(* IEC 61131-3 sources: material-handling-micro-cell/plc, 14 files *)

(* ---- FB_AlarmManager.st ---- *)
// ==========================================
// ALARM MANAGER MODULE FOR MHMC-01
// File: FB_AlarmManager.st
// Standard: IEC 61131-3 Structured Text
// Purpose: Alarm categorisation, acknowledgement, and stack light control.
// ==========================================

TYPE E_AlarmManagerState :
(
    ALARM_MGR_UNINITIALISED := 0,
    ALARM_MGR_NORMAL        := 10,
    ALARM_MGR_WARNING       := 20,
    ALARM_MGR_FAULT         := 30,
    ALARM_MGR_ABORT         := 900
) INT;
END_TYPE

TYPE E_MHMCAlarmCode :
(
    ALARM_NONE        := 0,
    ALARM_GENERAL_JAM := 100,
    ALARM_DIVERTER_1  := 200,
    ALARM_DIVERTER_2  := 210,
    ALARM_AIR_PRESSURE:= 300,
    ALARM_VFD_FAULT   := 400,
    ALARM_ESTOP       := 1000
) INT;
END_TYPE

TYPE ST_AlarmManagerConfig :
STRUCT
    rFlashPeriod_s : REAL; // Stack light flash interval.
END_STRUCT
END_TYPE

TYPE ST_AlarmManagerInput :
STRUCT
    xSafetyLoopOK       : BOOL;          // Safety relay input.
    xAirPressureOK      : BOOL;          // Pneumatic pressure healthy.
    xVfdFault           : BOOL;          // Conveyor drive fault.
    xJamAlarm           : BOOL;          // Jam detector alarm.
    xJamWarning         : BOOL;          // Jam detector pre-alarm.
    xDiverter1Faulted   : BOOL;          // Diverter 1 fault.
    xDiverter2Faulted   : BOOL;          // Diverter 2 fault.
    ePackMLState        : E_PackML_State; // Station state for light logic.
    xAcknowledge        : BOOL;          // HMI/SCADA alarm acknowledge.
    xReset              : BOOL;          // Alarm reset when root cause clear.
    rCycleTime_s        : REAL;          // PLC task interval for tests.
END_STRUCT
END_TYPE

TYPE ST_AlarmManagerOutput :
STRUCT
    xAnyAlarmActive     : BOOL;          // Aggregate active alarm.
    xAnyUnacked         : BOOL;          // Active or latched unacknowledged alarm.
    eActiveAlarmCode    : E_MHMCAlarmCode; // Highest-priority active alarm.
    uiSeverity          : UINT;          // OPC UA AlarmCondition severity 1..1000.
    xGeneralJamAlarm    : BOOL;          // OPC UA GeneralJamAlarm active state.
    xDiverter1Alarm     : BOOL;          // OPC UA Diverter1Fault active state.
    xDiverter2Alarm     : BOOL;          // OPC UA Diverter2Fault active state.
    xEStopAlarm         : BOOL;          // OPC UA EStopTripped active state.
    xStackGreen         : BOOL;          // Run indicator.
    xStackYellow        : BOOL;          // Warning/held indicator.
    xStackRed           : BOOL;          // Abort/fault indicator.
    xSounder            : BOOL;          // Audible alarm output.
    sActiveMessage      : STRING(80);    // Alarm text for SCADA.
END_STRUCT
END_TYPE

TYPE ST_AlarmManagerContext :
STRUCT
    eState          : E_AlarmManagerState;
    xInitialized    : BOOL;
    xAckLatched     : BOOL;
    xFlashState     : BOOL;
    rFlashElapsed_s : REAL;
END_STRUCT
END_TYPE

FUNCTION F_AlarmManager_Init : BOOL
VAR_INPUT
    stConfig : ST_AlarmManagerConfig;
END_VAR
VAR_IN_OUT
    stContext : ST_AlarmManagerContext;
    stOut     : ST_AlarmManagerOutput;
END_VAR

// Initialisation function. Clears latched acknowledgement and drives indicators safe.
stContext.eState := E_AlarmManagerState.ALARM_MGR_NORMAL;
stContext.xInitialized := TRUE;
stContext.xAckLatched := FALSE;
stContext.xFlashState := FALSE;
stContext.rFlashElapsed_s := 0.0;

stOut.xAnyAlarmActive := FALSE;
stOut.xAnyUnacked := FALSE;
stOut.eActiveAlarmCode := E_MHMCAlarmCode.ALARM_NONE;
stOut.uiSeverity := 0;
stOut.xGeneralJamAlarm := FALSE;
stOut.xDiverter1Alarm := FALSE;
stOut.xDiverter2Alarm := FALSE;
stOut.xEStopAlarm := FALSE;
stOut.xStackGreen := FALSE;
stOut.xStackYellow := FALSE;
stOut.xStackRed := FALSE;
stOut.xSounder := FALSE;
stOut.sActiveMessage := 'Alarm manager initialised';

F_AlarmManager_Init := TRUE;
END_FUNCTION

FUNCTION F_AlarmManager_Cyclic : BOOL
VAR_INPUT
    stIn     : ST_AlarmManagerInput;
    stConfig : ST_AlarmManagerConfig;
END_VAR
VAR_IN_OUT
    stContext : ST_AlarmManagerContext;
    stOut     : ST_AlarmManagerOutput;
END_VAR

// Cyclic execution function. Highest severity wins; acknowledgement is separated from reset.
stContext.rFlashElapsed_s := stContext.rFlashElapsed_s + stIn.rCycleTime_s;
IF stContext.rFlashElapsed_s >= stConfig.rFlashPeriod_s THEN
    stContext.xFlashState := NOT stContext.xFlashState;
    stContext.rFlashElapsed_s := 0.0;
END_IF;

stOut.xGeneralJamAlarm := stIn.xJamAlarm;
stOut.xDiverter1Alarm := stIn.xDiverter1Faulted;
stOut.xDiverter2Alarm := stIn.xDiverter2Faulted;
stOut.xEStopAlarm := NOT stIn.xSafetyLoopOK;
stOut.xAnyAlarmActive := stOut.xGeneralJamAlarm
                         OR stOut.xDiverter1Alarm
                         OR stOut.xDiverter2Alarm
                         OR stOut.xEStopAlarm
                         OR stIn.xVfdFault
                         OR NOT stIn.xAirPressureOK;

IF stIn.xAcknowledge THEN
    stContext.xAckLatched := TRUE;
END_IF;
IF stIn.xReset AND NOT stOut.xAnyAlarmActive THEN
    stContext.xAckLatched := FALSE;
END_IF;

IF NOT stContext.xInitialized THEN
    stContext.eState := E_AlarmManagerState.ALARM_MGR_UNINITIALISED;
    stOut.eActiveAlarmCode := E_MHMCAlarmCode.ALARM_NONE;
    stOut.uiSeverity := 0;
    stOut.sActiveMessage := 'Alarm manager not initialised';
ELSIF NOT stIn.xSafetyLoopOK THEN
    stContext.eState := E_AlarmManagerState.ALARM_MGR_ABORT;
    stOut.eActiveAlarmCode := E_MHMCAlarmCode.ALARM_ESTOP;
    stOut.uiSeverity := 1000;
    stOut.sActiveMessage := 'Emergency stop circuit tripped';
ELSIF stIn.xDiverter1Faulted THEN
    stContext.eState := E_AlarmManagerState.ALARM_MGR_FAULT;
    stOut.eActiveAlarmCode := E_MHMCAlarmCode.ALARM_DIVERTER_1;
    stOut.uiSeverity := 900;
    stOut.sActiveMessage := 'Diverter 1 pneumatic actuator fault';
ELSIF stIn.xDiverter2Faulted THEN
    stContext.eState := E_AlarmManagerState.ALARM_MGR_FAULT;
    stOut.eActiveAlarmCode := E_MHMCAlarmCode.ALARM_DIVERTER_2;
    stOut.uiSeverity := 900;
    stOut.sActiveMessage := 'Diverter 2 pneumatic actuator fault';
ELSIF stIn.xJamAlarm THEN
    stContext.eState := E_AlarmManagerState.ALARM_MGR_FAULT;
    stOut.eActiveAlarmCode := E_MHMCAlarmCode.ALARM_GENERAL_JAM;
    stOut.uiSeverity := 800;
    stOut.sActiveMessage := 'Package jam detected on main conveyor';
ELSIF NOT stIn.xAirPressureOK THEN
    stContext.eState := E_AlarmManagerState.ALARM_MGR_FAULT;
    stOut.eActiveAlarmCode := E_MHMCAlarmCode.ALARM_AIR_PRESSURE;
    stOut.uiSeverity := 700;
    stOut.sActiveMessage := 'Pneumatic pressure below permissive threshold';
ELSIF stIn.xVfdFault THEN
    stContext.eState := E_AlarmManagerState.ALARM_MGR_FAULT;
    stOut.eActiveAlarmCode := E_MHMCAlarmCode.ALARM_VFD_FAULT;
    stOut.uiSeverity := 700;
    stOut.sActiveMessage := 'Conveyor VFD fault active';
ELSIF stIn.xJamWarning OR (stIn.ePackMLState = E_PackML_State.HELD) THEN
    stContext.eState := E_AlarmManagerState.ALARM_MGR_WARNING;
    stOut.eActiveAlarmCode := E_MHMCAlarmCode.ALARM_NONE;
    stOut.uiSeverity := 300;
    stOut.sActiveMessage := 'Cell warning or held state active';
ELSE
    stContext.eState := E_AlarmManagerState.ALARM_MGR_NORMAL;
    stOut.eActiveAlarmCode := E_MHMCAlarmCode.ALARM_NONE;
    stOut.uiSeverity := 0;
    stOut.sActiveMessage := 'No active alarms';
END_IF;

stOut.xAnyUnacked := stOut.xAnyAlarmActive AND NOT stContext.xAckLatched;
stOut.xStackGreen := (stIn.ePackMLState = E_PackML_State.EXECUTE) AND NOT stOut.xAnyAlarmActive;
stOut.xStackYellow := stContext.xFlashState
                      AND ((stContext.eState = E_AlarmManagerState.ALARM_MGR_WARNING)
                           OR stIn.xJamWarning
                           OR stIn.xJamAlarm);
stOut.xStackRed := stOut.xEStopAlarm
                   OR (stContext.eState = E_AlarmManagerState.ALARM_MGR_FAULT)
                   OR (stContext.eState = E_AlarmManagerState.ALARM_MGR_ABORT);
stOut.xSounder := stOut.xAnyUnacked AND (stOut.uiSeverity >= 800);

F_AlarmManager_Cyclic := stContext.xInitialized;
END_FUNCTION

FUNCTION_BLOCK FB_AlarmManager
VAR_INPUT
    stIn     : ST_AlarmManagerInput;  // Typed symbolic inputs.
    stConfig : ST_AlarmManagerConfig; // Testable alarm configuration.
    xInit    : BOOL;                  // Pulse to re-run initialisation.
END_VAR
VAR_OUTPUT
    stOut        : ST_AlarmManagerOutput; // Typed symbolic outputs.
    eState       : E_AlarmManagerState;   // Exposed module state.
    xInitialized : BOOL;                  // Module initialisation complete.
END_VAR
VAR
    stContext : ST_AlarmManagerContext;
    xInitLast : BOOL;
END_VAR

IF (NOT stContext.xInitialized) OR (xInit AND NOT xInitLast) THEN
    F_AlarmManager_Init(stConfig := stConfig, stContext := stContext, stOut := stOut);
END_IF;

F_AlarmManager_Cyclic(stIn := stIn, stConfig := stConfig, stContext := stContext, stOut := stOut);

eState := stContext.eState;
xInitialized := stContext.xInitialized;
xInitLast := xInit;
END_FUNCTION_BLOCK

(* ---- FB_DiverterController.st ---- *)
// ==========================================
// DIVERTER CONTROLLER MODULE FOR MHMC-01
// File: FB_DiverterController.st
// Standard: IEC 61131-3 Structured Text
// Purpose: Pneumatic pusher sequencing for Diverter 1 and Diverter 2.
// ==========================================

TYPE E_DiverterControllerState :
(
    DIVERTER_UNINITIALISED := 0,
    DIVERTER_HOME          := 10,
    DIVERTER_EXTENDING     := 20,
    DIVERTER_WORK          := 30,
    DIVERTER_VERIFY        := 40,
    DIVERTER_RETRACTING    := 50,
    DIVERTER_FAULT         := 900
) INT;
END_TYPE

TYPE ST_DiverterControllerConfig :
STRUCT
    tActuatorName          : STRING(40); // Symbolic device name for diagnostics.
    rExtendTimeout_s       : REAL;       // Max time to reach work switch.
    rRetractTimeout_s      : REAL;       // Max time to return home.
    rWorkDwell_s           : REAL;       // Hold time after work switch.
    rVerificationTimeout_s : REAL;       // Max time to see lane PE confirmation.
END_STRUCT
END_TYPE

TYPE ST_DiverterControllerInput :
STRUCT
    xAutoEnable          : BOOL; // True when PackML EXECUTE permits automatic firing.
    xExtendRequest       : BOOL; // Routing sequence asks this diverter to fire.
    xManualExtend        : BOOL; // Maintenance/manual symbolic override.
    xHomeSensor          : BOOL; // LSx_Home magnetic switch.
    xWorkSensor          : BOOL; // LSx_Work magnetic switch.
    xVerificationSensor  : BOOL; // PE4 or PE5 lane confirmation.
    xResetFault          : BOOL; // Reset local actuator fault.
    rCycleTime_s         : REAL; // PLC task interval for test harness.
END_STRUCT
END_TYPE

TYPE ST_DiverterControllerOutput :
STRUCT
    xCommandExtend       : BOOL; // Symbolic solenoid command. Bind externally to field I/O.
    xBusy                : BOOL; // Actuator sequence active.
    xDone                : BOOL; // One-cycle sequence complete.
    xFaulted             : BOOL; // Travel or verification timeout.
    xHome                : BOOL; // Mirrored home switch.
    xWork                : BOOL; // Mirrored work switch.
    xVerified            : BOOL; // Lane verification latched for this cycle.
    uiFaultCode          : UINT; // 0 none, 1 extend, 2 retract, 3 verify.
    sStatusText          : STRING(80);
END_STRUCT
END_TYPE

TYPE ST_DiverterControllerContext :
STRUCT
    eState               : E_DiverterControllerState;
    xInitialized         : BOOL;
    xRequestLast         : BOOL;
    xDoneLatch           : BOOL;
    rStateElapsed_s      : REAL;
END_STRUCT
END_TYPE

FUNCTION F_DiverterController_Init : BOOL
VAR_INPUT
    stConfig : ST_DiverterControllerConfig;
END_VAR
VAR_IN_OUT
    stContext : ST_DiverterControllerContext;
    stOut     : ST_DiverterControllerOutput;
END_VAR

// Initialisation function. De-energises the valve and clears local sequence memory.
stContext.eState := E_DiverterControllerState.DIVERTER_HOME;
stContext.xInitialized := TRUE;
stContext.xRequestLast := FALSE;
stContext.xDoneLatch := FALSE;
stContext.rStateElapsed_s := 0.0;

stOut.xCommandExtend := FALSE;
stOut.xBusy := FALSE;
stOut.xDone := FALSE;
stOut.xFaulted := FALSE;
stOut.xHome := FALSE;
stOut.xWork := FALSE;
stOut.xVerified := FALSE;
stOut.uiFaultCode := 0;
stOut.sStatusText := 'Diverter controller initialised';

F_DiverterController_Init := TRUE;
END_FUNCTION

FUNCTION F_DiverterController_Cyclic : BOOL
VAR_INPUT
    stIn     : ST_DiverterControllerInput;
    stConfig : ST_DiverterControllerConfig;
END_VAR
VAR_IN_OUT
    stContext : ST_DiverterControllerContext;
    stOut     : ST_DiverterControllerOutput;
END_VAR
VAR
    xFireRequest : BOOL;
END_VAR

// Cyclic execution function. Sequence states are deterministic and unit-test friendly.
IF stIn.rCycleTime_s > 0.0 THEN
    stContext.rStateElapsed_s := stContext.rStateElapsed_s + stIn.rCycleTime_s;
END_IF;

stOut.xDone := FALSE;
stOut.xHome := stIn.xHomeSensor;
stOut.xWork := stIn.xWorkSensor;
xFireRequest := ((stIn.xAutoEnable AND stIn.xExtendRequest) OR stIn.xManualExtend);

IF stIn.xResetFault THEN
    stOut.xFaulted := FALSE;
    stOut.uiFaultCode := 0;
    stOut.xVerified := FALSE;
    stContext.eState := E_DiverterControllerState.DIVERTER_HOME;
    stContext.rStateElapsed_s := 0.0;
END_IF;

IF NOT stContext.xInitialized THEN
    stContext.eState := E_DiverterControllerState.DIVERTER_UNINITIALISED;
    stOut.xFaulted := TRUE;
    stOut.uiFaultCode := 99;
ELSIF stOut.xFaulted THEN
    stContext.eState := E_DiverterControllerState.DIVERTER_FAULT;
ELSIF xFireRequest AND NOT stContext.xRequestLast
      AND (stContext.eState = E_DiverterControllerState.DIVERTER_HOME) THEN
    stContext.eState := E_DiverterControllerState.DIVERTER_EXTENDING;
    stContext.rStateElapsed_s := 0.0;
    stOut.xVerified := FALSE;
ELSIF stContext.eState = E_DiverterControllerState.DIVERTER_EXTENDING THEN
    IF stIn.xWorkSensor THEN
        stContext.eState := E_DiverterControllerState.DIVERTER_WORK;
        stContext.rStateElapsed_s := 0.0;
    ELSIF stContext.rStateElapsed_s >= stConfig.rExtendTimeout_s THEN
        stOut.xFaulted := TRUE;
        stOut.uiFaultCode := 1;
    END_IF;
ELSIF stContext.eState = E_DiverterControllerState.DIVERTER_WORK THEN
    IF stContext.rStateElapsed_s >= stConfig.rWorkDwell_s THEN
        stContext.eState := E_DiverterControllerState.DIVERTER_VERIFY;
        stContext.rStateElapsed_s := 0.0;
    END_IF;
ELSIF stContext.eState = E_DiverterControllerState.DIVERTER_VERIFY THEN
    IF stIn.xVerificationSensor THEN
        stOut.xVerified := TRUE;
        stContext.eState := E_DiverterControllerState.DIVERTER_RETRACTING;
        stContext.rStateElapsed_s := 0.0;
    ELSIF stContext.rStateElapsed_s >= stConfig.rVerificationTimeout_s THEN
        stOut.xFaulted := TRUE;
        stOut.uiFaultCode := 3;
    END_IF;
ELSIF stContext.eState = E_DiverterControllerState.DIVERTER_RETRACTING THEN
    IF stIn.xHomeSensor THEN
        stContext.eState := E_DiverterControllerState.DIVERTER_HOME;
        stContext.rStateElapsed_s := 0.0;
        stOut.xDone := TRUE;
    ELSIF stContext.rStateElapsed_s >= stConfig.rRetractTimeout_s THEN
        stOut.xFaulted := TRUE;
        stOut.uiFaultCode := 2;
    END_IF;
ELSE
    stContext.eState := E_DiverterControllerState.DIVERTER_HOME;
END_IF;

stOut.xCommandExtend := (stContext.eState = E_DiverterControllerState.DIVERTER_EXTENDING)
                        OR (stContext.eState = E_DiverterControllerState.DIVERTER_WORK)
                        OR (stContext.eState = E_DiverterControllerState.DIVERTER_VERIFY);
stOut.xBusy := (stContext.eState = E_DiverterControllerState.DIVERTER_EXTENDING)
               OR (stContext.eState = E_DiverterControllerState.DIVERTER_WORK)
               OR (stContext.eState = E_DiverterControllerState.DIVERTER_VERIFY)
               OR (stContext.eState = E_DiverterControllerState.DIVERTER_RETRACTING);

IF stOut.xFaulted THEN
    stOut.xCommandExtend := FALSE;
    stOut.xBusy := FALSE;
    stOut.sStatusText := 'Diverter fault active';
ELSIF stOut.xBusy THEN
    stOut.sStatusText := 'Diverter sequence active';
ELSE
    stOut.sStatusText := 'Diverter ready at home';
END_IF;

stContext.xRequestLast := xFireRequest;
F_DiverterController_Cyclic := stContext.xInitialized;
END_FUNCTION

FUNCTION_BLOCK FB_DiverterController
VAR_INPUT
    stIn     : ST_DiverterControllerInput;  // Typed symbolic inputs.
    stConfig : ST_DiverterControllerConfig; // Testable timing configuration.
    xInit    : BOOL;                        // Pulse to re-run initialisation.
END_VAR
VAR_OUTPUT
    stOut        : ST_DiverterControllerOutput; // Typed symbolic outputs.
    eState       : E_DiverterControllerState;   // Exposed module state.
    xInitialized : BOOL;                        // Module initialisation complete.
END_VAR
VAR
    stContext : ST_DiverterControllerContext;
    xInitLast : BOOL;
END_VAR

IF (NOT stContext.xInitialized) OR (xInit AND NOT xInitLast) THEN
    F_DiverterController_Init(stConfig := stConfig, stContext := stContext, stOut := stOut);
END_IF;

F_DiverterController_Cyclic(stIn := stIn, stConfig := stConfig, stContext := stContext, stOut := stOut);

eState := stContext.eState;
xInitialized := stContext.xInitialized;
xInitLast := xInit;
END_FUNCTION_BLOCK

(* ---- FB_HistorianConnector.st ---- *)
// ==========================================
// HISTORIAN CONNECTOR MODULE FOR MHMC-01
// File: FB_HistorianConnector.st
// Standard: IEC 61131-3 Structured Text
// Purpose: PLC-side historian publish health and sampling handshake skeleton.
// ==========================================

TYPE E_HistorianConnectorState :
(
    HIST_UNINITIALISED := 0,
    HIST_DISABLED      := 10,
    HIST_CONNECTING    := 20,
    HIST_CONNECTED     := 30,
    HIST_PUBLISHING    := 40,
    HIST_BACKOFF       := 50,
    HIST_FAULTED       := 900
) INT;
END_TYPE

TYPE ST_HistorianConnectorConfig :
STRUCT
    tOpcUaNamespaceUri      : STRING(120); // Namespace URI, not an address binding.
    rSamplePeriod_s         : REAL;        // Historian sample strobe period.
    rHeartbeatTimeout_s     : REAL;        // Max time without collector heartbeat.
    uiMaxMissedHeartbeats   : UINT;        // Fault threshold.
END_STRUCT
END_TYPE

TYPE ST_HistorianConnectorInput :
STRUCT
    xEnable              : BOOL;               // Enable historian handshake.
    xOpcUaServerReady    : BOOL;               // OPC UA server namespace ready.
    xCollectorHeartbeat  : BOOL;               // Telegraf/collector heartbeat bit.
    xLastWriteOK         : BOOL;               // Influx write success from collector.
    stConveyor           : ST_Conveyor_Status; // Conveyor telemetry source.
    stDiverter1          : ST_Diverter_Status; // Diverter 1 telemetry source.
    stDiverter2          : ST_Diverter_Status; // Diverter 2 telemetry source.
    udiTotalCount        : UDINT;              // KPI source.
    udiLaneACount        : UDINT;              // KPI source.
    udiLaneBCount        : UDINT;              // KPI source.
    udiRejectCount       : UDINT;              // KPI source.
    uiTotalJams          : UINT;               // KPI source.
    rOEE_percent         : REAL;               // KPI source.
    xActiveAlarm         : BOOL;               // Alarm/event source.
    sActiveAlarmMessage  : STRING(80);         // Alarm/event source.
    rCycleTime_s         : REAL;               // PLC task interval for tests.
END_STRUCT
END_TYPE

TYPE ST_HistorianConnectorOutput :
STRUCT
    xSubscribeEnable      : BOOL;       // Allows collector to subscribe/poll OPC UA.
    xSampleStrobe         : BOOL;       // One-cycle sample request.
    xHistorianHealthy     : BOOL;       // True when OPC UA and collector are healthy.
    xPublishConveyor      : BOOL;       // Sample conveyor_telemetry.
    xPublishDiverter      : BOOL;       // Sample diverter_telemetry.
    xPublishKPI           : BOOL;       // Sample cell_kpis.
    xPublishAlarm         : BOOL;       // Sample alarms_events.
    uiMissedHeartbeats    : UINT;       // Collector heartbeat misses.
    sNamespaceUri         : STRING(120); // OPC UA namespace exposed to collector.
    sMeasurementClass     : STRING(40);  // Current logical measurement group.
    sLineProtocolPayload  : STRING(255); // Skeleton payload contract for collector tests.
    sStatusText           : STRING(80);
END_STRUCT
END_TYPE

TYPE ST_HistorianConnectorContext :
STRUCT
    eState             : E_HistorianConnectorState;
    xInitialized       : BOOL;
    xHeartbeatLast     : BOOL;
    rSampleElapsed_s   : REAL;
    rHeartbeatElapsed_s: REAL;
END_STRUCT
END_TYPE

FUNCTION F_HistorianConnector_Init : BOOL
VAR_INPUT
    stConfig : ST_HistorianConnectorConfig;
END_VAR
VAR_IN_OUT
    stContext : ST_HistorianConnectorContext;
    stOut     : ST_HistorianConnectorOutput;
END_VAR

// Initialisation function. The actual OPC UA/Influx endpoints remain external configuration.
stContext.eState := E_HistorianConnectorState.HIST_DISABLED;
stContext.xInitialized := TRUE;
stContext.xHeartbeatLast := FALSE;
stContext.rSampleElapsed_s := 0.0;
stContext.rHeartbeatElapsed_s := 0.0;

stOut.xSubscribeEnable := FALSE;
stOut.xSampleStrobe := FALSE;
stOut.xHistorianHealthy := FALSE;
stOut.xPublishConveyor := FALSE;
stOut.xPublishDiverter := FALSE;
stOut.xPublishKPI := FALSE;
stOut.xPublishAlarm := FALSE;
stOut.uiMissedHeartbeats := 0;
stOut.sNamespaceUri := stConfig.tOpcUaNamespaceUri;
stOut.sMeasurementClass := 'none';
stOut.sLineProtocolPayload := '';
stOut.sStatusText := 'Historian connector initialised';

F_HistorianConnector_Init := TRUE;
END_FUNCTION

FUNCTION F_HistorianConnector_Cyclic : BOOL
VAR_INPUT
    stIn     : ST_HistorianConnectorInput;
    stConfig : ST_HistorianConnectorConfig;
END_VAR
VAR_IN_OUT
    stContext : ST_HistorianConnectorContext;
    stOut     : ST_HistorianConnectorOutput;
END_VAR
VAR
    xHeartbeatEdge : BOOL;
END_VAR

// Cyclic execution function. Provides deterministic sample strobes for Telegraf/SCADA.
stOut.xSampleStrobe := FALSE;
stOut.xPublishConveyor := FALSE;
stOut.xPublishDiverter := FALSE;
stOut.xPublishKPI := FALSE;
stOut.xPublishAlarm := FALSE;
stOut.sNamespaceUri := stConfig.tOpcUaNamespaceUri;

xHeartbeatEdge := stIn.xCollectorHeartbeat <> stContext.xHeartbeatLast;
IF xHeartbeatEdge THEN
    stContext.rHeartbeatElapsed_s := 0.0;
    stOut.uiMissedHeartbeats := 0;
ELSE
    stContext.rHeartbeatElapsed_s := stContext.rHeartbeatElapsed_s + stIn.rCycleTime_s;
END_IF;

IF stContext.rHeartbeatElapsed_s >= stConfig.rHeartbeatTimeout_s THEN
    stOut.uiMissedHeartbeats := stOut.uiMissedHeartbeats + 1;
    stContext.rHeartbeatElapsed_s := 0.0;
END_IF;

IF NOT stContext.xInitialized THEN
    stContext.eState := E_HistorianConnectorState.HIST_UNINITIALISED;
ELSIF NOT stIn.xEnable THEN
    stContext.eState := E_HistorianConnectorState.HIST_DISABLED;
ELSIF NOT stIn.xOpcUaServerReady THEN
    stContext.eState := E_HistorianConnectorState.HIST_CONNECTING;
ELSIF stOut.uiMissedHeartbeats >= stConfig.uiMaxMissedHeartbeats THEN
    stContext.eState := E_HistorianConnectorState.HIST_BACKOFF;
ELSIF NOT stIn.xLastWriteOK THEN
    stContext.eState := E_HistorianConnectorState.HIST_FAULTED;
ELSE
    stContext.eState := E_HistorianConnectorState.HIST_CONNECTED;
END_IF;

stOut.xSubscribeEnable := stIn.xEnable AND stIn.xOpcUaServerReady;
stOut.xHistorianHealthy := stOut.xSubscribeEnable
                           AND (stOut.uiMissedHeartbeats < stConfig.uiMaxMissedHeartbeats)
                           AND stIn.xLastWriteOK;

IF stOut.xHistorianHealthy THEN
    stContext.rSampleElapsed_s := stContext.rSampleElapsed_s + stIn.rCycleTime_s;
    IF stContext.rSampleElapsed_s >= stConfig.rSamplePeriod_s THEN
        stContext.rSampleElapsed_s := 0.0;
        stContext.eState := E_HistorianConnectorState.HIST_PUBLISHING;
        stOut.xSampleStrobe := TRUE;
        stOut.xPublishConveyor := TRUE;
        stOut.xPublishDiverter := TRUE;
        stOut.xPublishKPI := TRUE;
        stOut.xPublishAlarm := stIn.xActiveAlarm;
    END_IF;
END_IF;

IF stOut.xPublishAlarm THEN
    stOut.sMeasurementClass := 'alarms_events';
    stOut.sLineProtocolPayload := 'alarms_events active=true';
ELSIF stOut.xPublishKPI THEN
    stOut.sMeasurementClass := 'cell_kpis';
    stOut.sLineProtocolPayload := 'cell_kpis sample=true';
ELSIF stOut.xPublishDiverter THEN
    stOut.sMeasurementClass := 'diverter_telemetry';
    stOut.sLineProtocolPayload := 'diverter_telemetry sample=true';
ELSIF stOut.xPublishConveyor THEN
    stOut.sMeasurementClass := 'conveyor_telemetry';
    stOut.sLineProtocolPayload := 'conveyor_telemetry sample=true';
ELSE
    stOut.sMeasurementClass := 'idle';
    stOut.sLineProtocolPayload := '';
END_IF;

IF stOut.xHistorianHealthy THEN
    stOut.sStatusText := 'Historian connector healthy';
ELSE
    stOut.sStatusText := 'Historian connector waiting for healthy collector';
END_IF;

stContext.xHeartbeatLast := stIn.xCollectorHeartbeat;
F_HistorianConnector_Cyclic := stContext.xInitialized;
END_FUNCTION

FUNCTION_BLOCK FB_HistorianConnector
VAR_INPUT
    stIn     : ST_HistorianConnectorInput;  // Typed symbolic inputs.
    stConfig : ST_HistorianConnectorConfig; // Testable historian configuration.
    xInit    : BOOL;                        // Pulse to re-run initialisation.
END_VAR
VAR_OUTPUT
    stOut        : ST_HistorianConnectorOutput; // Typed symbolic outputs.
    eState       : E_HistorianConnectorState;   // Exposed module state.
    xInitialized : BOOL;                        // Module initialisation complete.
END_VAR
VAR
    stContext : ST_HistorianConnectorContext;
    xInitLast : BOOL;
END_VAR

IF (NOT stContext.xInitialized) OR (xInit AND NOT xInitLast) THEN
    F_HistorianConnector_Init(stConfig := stConfig, stContext := stContext, stOut := stOut);
END_IF;

F_HistorianConnector_Cyclic(stIn := stIn, stConfig := stConfig, stContext := stContext, stOut := stOut);

eState := stContext.eState;
xInitialized := stContext.xInitialized;
xInitLast := xInit;
END_FUNCTION_BLOCK

(* ---- FB_JamDetector.st ---- *)
// ==========================================
// JAM DETECTOR MODULE FOR MHMC-01
// File: FB_JamDetector.st
// Standard: IEC 61131-3 Structured Text
// Purpose: Dynamic PE1/PE2/PE3 blockage watchdogs.
// ==========================================

TYPE E_JamDetectorState :
(
    JAM_DET_UNINITIALISED := 0,
    JAM_DET_CLEAR         := 10,
    JAM_DET_MONITORING    := 20,
    JAM_DET_WARNING       := 30,
    JAM_DET_JAMMED        := 900
) INT;
END_TYPE

TYPE ST_JamDetectorConfig :
STRUCT
    rReferenceSpeed_mps : REAL; // Speed used for nominal 3.0 s FDS limit.
    rBaseJamLimit_s     : REAL; // Nominal jam threshold at reference speed.
    rMaximumJamLimit_s  : REAL; // Slow-speed upper watchdog bound.
    rWarningRatio       : REAL; // Warning before full jam, e.g. 0.80.
END_STRUCT
END_TYPE

TYPE ST_JamDetectorInput :
STRUCT
    xRawPE1            : BOOL; // PE1 infeed blocked.
    xRawPE2            : BOOL; // PE2 scan trigger blocked.
    xRawPE3            : BOOL; // PE3 diverter in-range blocked.
    xConveyorRunning   : BOOL; // Conveyor feedback.
    rConveyorSpeed_mps : REAL; // Conveyor feedback speed.
    xResetJam          : BOOL; // ResetJam RPC/HMI command.
    rCycleTime_s       : REAL; // PLC task interval for unit tests.
END_STRUCT
END_TYPE

TYPE ST_JamDetectorOutput :
STRUCT
    xJamAlarm          : BOOL; // Fault flag to StationController.
    xWarning           : BOOL; // Pre-alarm for HMI and beacon logic.
    xBeaconYellowFlash : BOOL; // Symbolic stack light request.
    uiJamSource        : UINT; // 0 none, 1 PE1, 2 PE2, 3 PE3.
    uiTotalJams        : UINT; // OPC UA KPI TotalJams node.
    rActiveLimit_s     : REAL; // Dynamic watchdog threshold in use.
    sStatusText        : STRING(80);
END_STRUCT
END_TYPE

TYPE ST_JamDetectorContext :
STRUCT
    eState          : E_JamDetectorState;
    xInitialized    : BOOL;
    xJamLatchedLast : BOOL;
    rPE1Blocked_s   : REAL;
    rPE2Blocked_s   : REAL;
    rPE3Blocked_s   : REAL;
END_STRUCT
END_TYPE

FUNCTION F_JamDetector_DynamicLimit_s : REAL
VAR_INPUT
    rConveyorSpeed_mps : REAL;
    stConfig           : ST_JamDetectorConfig;
END_VAR
VAR
    rLimit_s : REAL;
END_VAR

// Dynamic limit increases as conveyor speed drops. It is clamped for slow jog cases.
IF rConveyorSpeed_mps <= 0.01 THEN
    rLimit_s := stConfig.rMaximumJamLimit_s;
ELSE
    rLimit_s := stConfig.rBaseJamLimit_s * stConfig.rReferenceSpeed_mps / rConveyorSpeed_mps;
END_IF;

IF rLimit_s < stConfig.rBaseJamLimit_s THEN
    rLimit_s := stConfig.rBaseJamLimit_s;
END_IF;
IF rLimit_s > stConfig.rMaximumJamLimit_s THEN
    rLimit_s := stConfig.rMaximumJamLimit_s;
END_IF;

F_JamDetector_DynamicLimit_s := rLimit_s;
END_FUNCTION

FUNCTION F_JamDetector_Init : BOOL
VAR_INPUT
    stConfig : ST_JamDetectorConfig;
END_VAR
VAR_IN_OUT
    stContext : ST_JamDetectorContext;
    stOut     : ST_JamDetectorOutput;
END_VAR

// Initialisation function. Clears watchdog accumulators and alarm outputs.
stContext.eState := E_JamDetectorState.JAM_DET_CLEAR;
stContext.xInitialized := TRUE;
stContext.xJamLatchedLast := FALSE;
stContext.rPE1Blocked_s := 0.0;
stContext.rPE2Blocked_s := 0.0;
stContext.rPE3Blocked_s := 0.0;

stOut.xJamAlarm := FALSE;
stOut.xWarning := FALSE;
stOut.xBeaconYellowFlash := FALSE;
stOut.uiJamSource := 0;
stOut.uiTotalJams := 0;
stOut.rActiveLimit_s := stConfig.rBaseJamLimit_s;
stOut.sStatusText := 'Jam detector initialised';

F_JamDetector_Init := TRUE;
END_FUNCTION

FUNCTION F_JamDetector_Cyclic : BOOL
VAR_INPUT
    stIn     : ST_JamDetectorInput;
    stConfig : ST_JamDetectorConfig;
END_VAR
VAR_IN_OUT
    stContext : ST_JamDetectorContext;
    stOut     : ST_JamDetectorOutput;
END_VAR
VAR
    rWarnLimit_s : REAL;
    xAnyBlocked  : BOOL;
END_VAR

// Cyclic execution function. PE watchdogs are independent and symbolic.
stOut.rActiveLimit_s := F_JamDetector_DynamicLimit_s(rConveyorSpeed_mps := stIn.rConveyorSpeed_mps, stConfig := stConfig);
rWarnLimit_s := stOut.rActiveLimit_s * stConfig.rWarningRatio;
xAnyBlocked := stIn.xRawPE1 OR stIn.xRawPE2 OR stIn.xRawPE3;

IF stIn.xResetJam THEN
    stOut.xJamAlarm := FALSE;
    stOut.xWarning := FALSE;
    stOut.xBeaconYellowFlash := FALSE;
    stOut.uiJamSource := 0;
    stContext.rPE1Blocked_s := 0.0;
    stContext.rPE2Blocked_s := 0.0;
    stContext.rPE3Blocked_s := 0.0;
    stContext.eState := E_JamDetectorState.JAM_DET_CLEAR;
END_IF;

IF stIn.xConveyorRunning THEN
    IF stIn.xRawPE1 THEN
        stContext.rPE1Blocked_s := stContext.rPE1Blocked_s + stIn.rCycleTime_s;
    ELSE
        stContext.rPE1Blocked_s := 0.0;
    END_IF;

    IF stIn.xRawPE2 THEN
        stContext.rPE2Blocked_s := stContext.rPE2Blocked_s + stIn.rCycleTime_s;
    ELSE
        stContext.rPE2Blocked_s := 0.0;
    END_IF;

    IF stIn.xRawPE3 THEN
        stContext.rPE3Blocked_s := stContext.rPE3Blocked_s + stIn.rCycleTime_s;
    ELSE
        stContext.rPE3Blocked_s := 0.0;
    END_IF;
END_IF;

IF NOT stContext.xInitialized THEN
    stContext.eState := E_JamDetectorState.JAM_DET_UNINITIALISED;
ELSIF (stContext.rPE1Blocked_s >= stOut.rActiveLimit_s)
      OR (stContext.rPE2Blocked_s >= stOut.rActiveLimit_s)
      OR (stContext.rPE3Blocked_s >= stOut.rActiveLimit_s) THEN
    stContext.eState := E_JamDetectorState.JAM_DET_JAMMED;
    stOut.xJamAlarm := TRUE;
    IF stContext.rPE1Blocked_s >= stOut.rActiveLimit_s THEN
        stOut.uiJamSource := 1;
    ELSIF stContext.rPE2Blocked_s >= stOut.rActiveLimit_s THEN
        stOut.uiJamSource := 2;
    ELSE
        stOut.uiJamSource := 3;
    END_IF;
ELSIF (stContext.rPE1Blocked_s >= rWarnLimit_s)
      OR (stContext.rPE2Blocked_s >= rWarnLimit_s)
      OR (stContext.rPE3Blocked_s >= rWarnLimit_s) THEN
    stContext.eState := E_JamDetectorState.JAM_DET_WARNING;
    stOut.xWarning := TRUE;
ELSE
    stOut.xWarning := FALSE;
    IF xAnyBlocked AND stIn.xConveyorRunning THEN
        stContext.eState := E_JamDetectorState.JAM_DET_MONITORING;
    ELSE
        stContext.eState := E_JamDetectorState.JAM_DET_CLEAR;
    END_IF;
END_IF;

IF stOut.xJamAlarm AND NOT stContext.xJamLatchedLast THEN
    stOut.uiTotalJams := stOut.uiTotalJams + 1;
END_IF;

stOut.xBeaconYellowFlash := stOut.xWarning OR stOut.xJamAlarm;
IF stOut.xJamAlarm THEN
    stOut.sStatusText := 'Package jam detected on main conveyor';
ELSIF stOut.xWarning THEN
    stOut.sStatusText := 'Photoeye blocked near jam threshold';
ELSE
    stOut.sStatusText := 'Jam detector clear';
END_IF;

stContext.xJamLatchedLast := stOut.xJamAlarm;
F_JamDetector_Cyclic := stContext.xInitialized;
END_FUNCTION

FUNCTION_BLOCK FB_JamDetector
VAR_INPUT
    stIn     : ST_JamDetectorInput;  // Typed symbolic inputs.
    stConfig : ST_JamDetectorConfig; // Testable watchdog configuration.
    xInit    : BOOL;                 // Pulse to re-run initialisation.
END_VAR
VAR_OUTPUT
    stOut        : ST_JamDetectorOutput; // Typed symbolic outputs.
    eState       : E_JamDetectorState;   // Exposed module state.
    xInitialized : BOOL;                 // Module initialisation complete.
END_VAR
VAR
    stContext : ST_JamDetectorContext;
    xInitLast : BOOL;
END_VAR

IF (NOT stContext.xInitialized) OR (xInit AND NOT xInitLast) THEN
    F_JamDetector_Init(stConfig := stConfig, stContext := stContext, stOut := stOut);
END_IF;

F_JamDetector_Cyclic(stIn := stIn, stConfig := stConfig, stContext := stContext, stOut := stOut);

eState := stContext.eState;
xInitialized := stContext.xInitialized;
xInitLast := xInit;
END_FUNCTION_BLOCK

(* ---- FB_KPIService.st ---- *)
// ==========================================
// KPI SERVICE MODULE FOR MHMC-01
// File: FB_KPIService.st
// Standard: IEC 61131-3 Structured Text
// Purpose: Throughput counters and OEE calculation skeleton.
// ==========================================

TYPE E_KPIServiceState :
(
    KPI_UNINITIALISED := 0,
    KPI_IDLE          := 10,
    KPI_ACCUMULATING  := 20,
    KPI_HELD          := 30,
    KPI_RESETTING     := 40
) INT;
END_TYPE

TYPE ST_KPIServiceConfig :
STRUCT
    rPerformanceFactor : REAL; // FDS target sorting velocity efficiency, e.g. 0.96.
    rTargetRate_ppm    : REAL; // Target packages per minute for throughput trending.
END_STRUCT
END_TYPE

TYPE ST_KPIServiceInput :
STRUCT
    xPE4LaneA        : BOOL;          // Lane A verification sensor.
    xPE5LaneB        : BOOL;          // Lane B verification sensor.
    xPE6Reject       : BOOL;          // Reject verification sensor.
    ePackMLState     : E_PackML_State; // Station state for availability.
    xFaultDowntime   : BOOL;          // Fault/held downtime active.
    xResetCounters   : BOOL;          // KPI reset command.
    rCycleTime_s     : REAL;          // PLC task interval for tests.
END_STRUCT
END_TYPE

TYPE ST_KPIServiceOutput :
STRUCT
    udiTotalPackages     : UDINT; // Total package count.
    udiLaneAPackages     : UDINT; // Lane A count.
    udiLaneBPackages     : UDINT; // Lane B count.
    udiRejectPackages    : UDINT; // Reject count.
    rAvailability        : REAL;  // Execute / scheduled time.
    rPerformance         : REAL;  // Target sorting velocity efficiency.
    rQuality             : REAL;  // (Total - Reject) / Total.
    rOEE_percent         : REAL;  // Availability * Performance * Quality * 100.
    rThroughput_ppm      : REAL;  // Recent average from total/scheduled time.
    sStatusText          : STRING(80);
END_STRUCT
END_TYPE

TYPE ST_KPIServiceContext :
STRUCT
    eState            : E_KPIServiceState;
    xInitialized      : BOOL;
    xPE4Last          : BOOL;
    xPE5Last          : BOOL;
    xPE6Last          : BOOL;
    rExecuteTime_s    : REAL;
    rFaultDowntime_s  : REAL;
    rScheduledTime_s  : REAL;
END_STRUCT
END_TYPE

FUNCTION F_KPIService_Init : BOOL
VAR_INPUT
    stConfig : ST_KPIServiceConfig;
END_VAR
VAR_IN_OUT
    stContext : ST_KPIServiceContext;
    stOut     : ST_KPIServiceOutput;
END_VAR

// Initialisation function. Clears counters and restores default OEE factors.
stContext.eState := E_KPIServiceState.KPI_IDLE;
stContext.xInitialized := TRUE;
stContext.xPE4Last := FALSE;
stContext.xPE5Last := FALSE;
stContext.xPE6Last := FALSE;
stContext.rExecuteTime_s := 0.0;
stContext.rFaultDowntime_s := 0.0;
stContext.rScheduledTime_s := 0.0;

stOut.udiTotalPackages := 0;
stOut.udiLaneAPackages := 0;
stOut.udiLaneBPackages := 0;
stOut.udiRejectPackages := 0;
stOut.rAvailability := 1.0;
stOut.rPerformance := stConfig.rPerformanceFactor;
stOut.rQuality := 1.0;
stOut.rOEE_percent := stOut.rAvailability * stOut.rPerformance * stOut.rQuality * 100.0;
stOut.rThroughput_ppm := 0.0;
stOut.sStatusText := 'KPI service initialised';

F_KPIService_Init := TRUE;
END_FUNCTION

FUNCTION F_KPIService_Cyclic : BOOL
VAR_INPUT
    stIn     : ST_KPIServiceInput;
    stConfig : ST_KPIServiceConfig;
END_VAR
VAR_IN_OUT
    stContext : ST_KPIServiceContext;
    stOut     : ST_KPIServiceOutput;
END_VAR
VAR
    xPE4Rise : BOOL;
    xPE5Rise : BOOL;
    xPE6Rise : BOOL;
END_VAR

// Cyclic execution function. Sensor edges drive counters; PackML state drives availability.
IF stIn.xResetCounters THEN
    stContext.eState := E_KPIServiceState.KPI_RESETTING;
    stContext.rExecuteTime_s := 0.0;
    stContext.rFaultDowntime_s := 0.0;
    stContext.rScheduledTime_s := 0.0;
    stOut.udiTotalPackages := 0;
    stOut.udiLaneAPackages := 0;
    stOut.udiLaneBPackages := 0;
    stOut.udiRejectPackages := 0;
END_IF;

xPE4Rise := stIn.xPE4LaneA AND NOT stContext.xPE4Last;
xPE5Rise := stIn.xPE5LaneB AND NOT stContext.xPE5Last;
xPE6Rise := stIn.xPE6Reject AND NOT stContext.xPE6Last;

IF xPE4Rise THEN
    stOut.udiLaneAPackages := stOut.udiLaneAPackages + 1;
    stOut.udiTotalPackages := stOut.udiTotalPackages + 1;
END_IF;
IF xPE5Rise THEN
    stOut.udiLaneBPackages := stOut.udiLaneBPackages + 1;
    stOut.udiTotalPackages := stOut.udiTotalPackages + 1;
END_IF;
IF xPE6Rise THEN
    stOut.udiRejectPackages := stOut.udiRejectPackages + 1;
    stOut.udiTotalPackages := stOut.udiTotalPackages + 1;
END_IF;

IF stIn.ePackMLState = E_PackML_State.EXECUTE THEN
    stContext.eState := E_KPIServiceState.KPI_ACCUMULATING;
    stContext.rExecuteTime_s := stContext.rExecuteTime_s + stIn.rCycleTime_s;
    stContext.rScheduledTime_s := stContext.rScheduledTime_s + stIn.rCycleTime_s;
ELSIF stIn.xFaultDowntime OR (stIn.ePackMLState = E_PackML_State.HELD) THEN
    stContext.eState := E_KPIServiceState.KPI_HELD;
    stContext.rFaultDowntime_s := stContext.rFaultDowntime_s + stIn.rCycleTime_s;
    stContext.rScheduledTime_s := stContext.rScheduledTime_s + stIn.rCycleTime_s;
ELSE
    stContext.eState := E_KPIServiceState.KPI_IDLE;
END_IF;

IF stContext.rScheduledTime_s > 0.0 THEN
    stOut.rAvailability := stContext.rExecuteTime_s / stContext.rScheduledTime_s;
    stOut.rThroughput_ppm := UDINT_TO_REAL(stOut.udiTotalPackages) / (stContext.rScheduledTime_s / 60.0);
ELSE
    stOut.rAvailability := 1.0;
    stOut.rThroughput_ppm := 0.0;
END_IF;

stOut.rPerformance := stConfig.rPerformanceFactor;
IF stOut.udiTotalPackages > 0 THEN
    stOut.rQuality := (UDINT_TO_REAL(stOut.udiTotalPackages) - UDINT_TO_REAL(stOut.udiRejectPackages))
                      / UDINT_TO_REAL(stOut.udiTotalPackages);
ELSE
    stOut.rQuality := 1.0;
END_IF;

stOut.rOEE_percent := stOut.rAvailability * stOut.rPerformance * stOut.rQuality * 100.0;
stOut.sStatusText := 'KPI service calculated counters and OEE';

stContext.xPE4Last := stIn.xPE4LaneA;
stContext.xPE5Last := stIn.xPE5LaneB;
stContext.xPE6Last := stIn.xPE6Reject;
F_KPIService_Cyclic := stContext.xInitialized;
END_FUNCTION

FUNCTION_BLOCK FB_KPIService
VAR_INPUT
    stIn     : ST_KPIServiceInput;  // Typed symbolic inputs.
    stConfig : ST_KPIServiceConfig; // Testable KPI configuration.
    xInit    : BOOL;                // Pulse to re-run initialisation.
END_VAR
VAR_OUTPUT
    stOut        : ST_KPIServiceOutput; // Typed symbolic outputs.
    eState       : E_KPIServiceState;   // Exposed module state.
    xInitialized : BOOL;                // Module initialisation complete.
END_VAR
VAR
    stContext : ST_KPIServiceContext;
    xInitLast : BOOL;
END_VAR

IF (NOT stContext.xInitialized) OR (xInit AND NOT xInitLast) THEN
    F_KPIService_Init(stConfig := stConfig, stContext := stContext, stOut := stOut);
END_IF;

F_KPIService_Cyclic(stIn := stIn, stConfig := stConfig, stContext := stContext, stOut := stOut);

eState := stContext.eState;
xInitialized := stContext.xInitialized;
xInitLast := xInit;
END_FUNCTION_BLOCK

(* ---- FB_LineSupervisor.st ---- *)
// ==========================================
// LINE SUPERVISOR MODULE FOR MHMC-01
// File: FB_LineSupervisor.st
// Standard: IEC 61131-3 Structured Text
// Purpose: Cell-level command, mode, and recipe dispatch skeleton.
// ==========================================

TYPE E_LineSupervisorState :
(
    LINE_SUP_UNINITIALISED := 0,
    LINE_SUP_READY         := 10,
    LINE_SUP_RECIPE_LOAD   := 20,
    LINE_SUP_COMMANDING    := 30,
    LINE_SUP_FAULTED       := 900
) INT;
END_TYPE

TYPE ST_LineSupervisorConfig :
STRUCT
    rDefaultTargetSpeed_mps : REAL;       // Recipe default conveyor speed.
    rMinimumTargetSpeed_mps : REAL;       // Lower recipe validation bound.
    rMaximumTargetSpeed_mps : REAL;       // Upper recipe validation bound.
    sLaneAPattern           : STRING(40); // Symbolic barcode rule for Lane A.
    sLaneBPattern           : STRING(40); // Symbolic barcode rule for Lane B.
    sRejectPattern          : STRING(40); // Symbolic barcode rule for reject/default.
END_STRUCT
END_TYPE

TYPE ST_LineSupervisorInput :
STRUCT
    xStartCommand      : BOOL;          // HMI/OPC UA StartCell request.
    xStopCommand       : BOOL;          // HMI/OPC UA StopCell request.
    xResetCommand      : BOOL;          // HMI/OPC UA reset request.
    xHoldCommand       : BOOL;          // HMI/SCADA hold request.
    xUnholdCommand     : BOOL;          // HMI/SCADA unhold request.
    xClearCommand      : BOOL;          // Clear aborted state request.
    xLoadRecipeCommand : BOOL;          // HMI/OPC UA LoadRecipe request.
    uiRecipeSelect     : UINT;          // Symbolic recipe selector.
    rRecipeSpeed_mps   : REAL;          // Recipe speed requested by supervisor.
    eModeSelect        : E_PackML_Mode; // Requested PackML operating mode.
    xOpcUaConnected    : BOOL;          // Supervisory channel healthy.
    xStationReady      : BOOL;          // Station can accept supervisor commands.
END_STRUCT
END_TYPE

TYPE ST_LineSupervisorOutput :
STRUCT
    xStartCellPulse     : BOOL;          // One-cycle StartCell command.
    xStopCellPulse      : BOOL;          // One-cycle StopCell command.
    xResetCellPulse     : BOOL;          // One-cycle reset command.
    xHoldCell           : BOOL;          // Level hold command.
    xUnholdCellPulse    : BOOL;          // One-cycle unhold command.
    xClearCellPulse     : BOOL;          // One-cycle clear command.
    xLoadRecipePulse    : BOOL;          // One-cycle recipe load command.
    eRequestedMode      : E_PackML_Mode; // Mode written to ControlState.CurrentMode.
    uiActiveRecipe      : UINT;          // Accepted recipe ID.
    rTargetSpeed_mps    : REAL;          // Recipe speed dispatched to station.
    sLaneAPattern       : STRING(40);    // Dispatch barcode rule for Lane A.
    sLaneBPattern       : STRING(40);    // Dispatch barcode rule for Lane B.
    sRejectPattern      : STRING(40);    // Dispatch barcode rule for Reject.
    xRecipeValid        : BOOL;          // Recipe parameters accepted.
    xSupervisorHealthy  : BOOL;          // True when command channel and recipe are valid.
    sStatusText         : STRING(80);    // Diagnostic text for HMI/OPC UA.
END_STRUCT
END_TYPE

TYPE ST_LineSupervisorContext :
STRUCT
    eState              : E_LineSupervisorState;
    xInitialized        : BOOL;
    xStartLast          : BOOL;
    xStopLast           : BOOL;
    xResetLast          : BOOL;
    xUnholdLast         : BOOL;
    xClearLast          : BOOL;
    xLoadRecipeLast     : BOOL;
END_STRUCT
END_TYPE

FUNCTION F_LineSupervisor_Init : BOOL
VAR_INPUT
    stConfig : ST_LineSupervisorConfig;
END_VAR
VAR_IN_OUT
    stContext : ST_LineSupervisorContext;
    stOut     : ST_LineSupervisorOutput;
END_VAR

// Initialisation function. Unit tests can call this directly before exercising Cyclic.
stContext.eState := E_LineSupervisorState.LINE_SUP_READY;
stContext.xInitialized := TRUE;
stContext.xStartLast := FALSE;
stContext.xStopLast := FALSE;
stContext.xResetLast := FALSE;
stContext.xUnholdLast := FALSE;
stContext.xClearLast := FALSE;
stContext.xLoadRecipeLast := FALSE;

stOut.xStartCellPulse := FALSE;
stOut.xStopCellPulse := FALSE;
stOut.xResetCellPulse := FALSE;
stOut.xHoldCell := FALSE;
stOut.xUnholdCellPulse := FALSE;
stOut.xClearCellPulse := FALSE;
stOut.xLoadRecipePulse := FALSE;
stOut.eRequestedMode := E_PackML_Mode.AUTO;
stOut.uiActiveRecipe := 0;
stOut.rTargetSpeed_mps := stConfig.rDefaultTargetSpeed_mps;
stOut.sLaneAPattern := stConfig.sLaneAPattern;
stOut.sLaneBPattern := stConfig.sLaneBPattern;
stOut.sRejectPattern := stConfig.sRejectPattern;
stOut.xRecipeValid := TRUE;
stOut.xSupervisorHealthy := TRUE;
stOut.sStatusText := 'Line supervisor initialised';

F_LineSupervisor_Init := TRUE;
END_FUNCTION

FUNCTION F_LineSupervisor_Cyclic : BOOL
VAR_INPUT
    stIn     : ST_LineSupervisorInput;
    stConfig : ST_LineSupervisorConfig;
END_VAR
VAR_IN_OUT
    stContext : ST_LineSupervisorContext;
    stOut     : ST_LineSupervisorOutput;
END_VAR
VAR
    xSpeedInsideLimits : BOOL;
END_VAR

// Cyclic execution function. All I/O is symbolic and supplied through typed structures.
stOut.xStartCellPulse := FALSE;
stOut.xStopCellPulse := FALSE;
stOut.xResetCellPulse := FALSE;
stOut.xUnholdCellPulse := FALSE;
stOut.xClearCellPulse := FALSE;
stOut.xLoadRecipePulse := FALSE;
stOut.xHoldCell := stIn.xHoldCommand;
stOut.eRequestedMode := stIn.eModeSelect;

xSpeedInsideLimits := (stIn.rRecipeSpeed_mps >= stConfig.rMinimumTargetSpeed_mps)
                      AND (stIn.rRecipeSpeed_mps <= stConfig.rMaximumTargetSpeed_mps);

IF NOT stContext.xInitialized THEN
    stContext.eState := E_LineSupervisorState.LINE_SUP_UNINITIALISED;
    stOut.xSupervisorHealthy := FALSE;
    stOut.sStatusText := 'Line supervisor not initialised';
ELSIF NOT stIn.xOpcUaConnected THEN
    stContext.eState := E_LineSupervisorState.LINE_SUP_FAULTED;
    stOut.xSupervisorHealthy := FALSE;
    stOut.sStatusText := 'OPC UA supervisory channel not healthy';
ELSIF stIn.xLoadRecipeCommand AND NOT stContext.xLoadRecipeLast THEN
    stContext.eState := E_LineSupervisorState.LINE_SUP_RECIPE_LOAD;
    stOut.xLoadRecipePulse := TRUE;
    stOut.xRecipeValid := xSpeedInsideLimits;
    IF xSpeedInsideLimits THEN
        stOut.uiActiveRecipe := stIn.uiRecipeSelect;
        stOut.rTargetSpeed_mps := stIn.rRecipeSpeed_mps;
        stOut.sLaneAPattern := stConfig.sLaneAPattern;
        stOut.sLaneBPattern := stConfig.sLaneBPattern;
        stOut.sRejectPattern := stConfig.sRejectPattern;
        stOut.xSupervisorHealthy := TRUE;
        stOut.sStatusText := 'Recipe accepted and dispatched';
    ELSE
        stContext.eState := E_LineSupervisorState.LINE_SUP_FAULTED;
        stOut.xSupervisorHealthy := FALSE;
        stOut.sStatusText := 'Recipe speed outside configured limits';
    END_IF;
ELSIF stIn.xStationReady THEN
    stContext.eState := E_LineSupervisorState.LINE_SUP_COMMANDING;
    stOut.xStartCellPulse := stIn.xStartCommand AND NOT stContext.xStartLast;
    stOut.xStopCellPulse := stIn.xStopCommand AND NOT stContext.xStopLast;
    stOut.xResetCellPulse := stIn.xResetCommand AND NOT stContext.xResetLast;
    stOut.xUnholdCellPulse := stIn.xUnholdCommand AND NOT stContext.xUnholdLast;
    stOut.xClearCellPulse := stIn.xClearCommand AND NOT stContext.xClearLast;
    stOut.xSupervisorHealthy := stOut.xRecipeValid;
    stOut.sStatusText := 'Supervisor command interface ready';
ELSE
    stContext.eState := E_LineSupervisorState.LINE_SUP_READY;
    stOut.xSupervisorHealthy := stOut.xRecipeValid;
    stOut.sStatusText := 'Waiting for station ready';
END_IF;

stContext.xStartLast := stIn.xStartCommand;
stContext.xStopLast := stIn.xStopCommand;
stContext.xResetLast := stIn.xResetCommand;
stContext.xUnholdLast := stIn.xUnholdCommand;
stContext.xClearLast := stIn.xClearCommand;
stContext.xLoadRecipeLast := stIn.xLoadRecipeCommand;

F_LineSupervisor_Cyclic := stContext.xInitialized;
END_FUNCTION

FUNCTION_BLOCK FB_LineSupervisor
VAR_INPUT
    stIn     : ST_LineSupervisorInput;  // Typed symbolic inputs.
    stConfig : ST_LineSupervisorConfig; // Testable configuration.
    xInit    : BOOL;                    // Pulse to re-run initialisation.
END_VAR
VAR_OUTPUT
    stOut        : ST_LineSupervisorOutput; // Typed symbolic outputs.
    eState       : E_LineSupervisorState;   // Exposed module state.
    xInitialized : BOOL;                    // Module initialisation complete.
END_VAR
VAR
    stContext : ST_LineSupervisorContext;
    xInitLast : BOOL;
END_VAR

// FB wrapper: call this POU every PLC task cycle, or call Init/Cyclic functions directly in tests.
IF (NOT stContext.xInitialized) OR (xInit AND NOT xInitLast) THEN
    F_LineSupervisor_Init(stConfig := stConfig, stContext := stContext, stOut := stOut);
END_IF;

F_LineSupervisor_Cyclic(stIn := stIn, stConfig := stConfig, stContext := stContext, stOut := stOut);

eState := stContext.eState;
xInitialized := stContext.xInitialized;
xInitLast := xInit;
END_FUNCTION_BLOCK

(* ---- FB_StationController.st ---- *)
// ==========================================
// STATION CONTROLLER MODULE FOR MHMC-01
// File: FB_StationController.st
// Standard: IEC 61131-3 Structured Text
// Purpose: PackML station control and symbolic PLCopen motion command adapter.
// ==========================================

TYPE E_StationControllerState :
(
    STATION_UNINITIALISED := 0,
    STATION_STOPPED       := 10,
    STATION_RESETTING     := 20,
    STATION_IDLE          := 30,
    STATION_STARTING      := 40,
    STATION_EXECUTE       := 50,
    STATION_SUSPENDED     := 60,
    STATION_HOLDING       := 70,
    STATION_HELD          := 80,
    STATION_UNHOLDING     := 90,
    STATION_STOPPING      := 100,
    STATION_ABORTED       := 900
) INT;
END_TYPE

TYPE ST_PLCopenMotionCommand :
STRUCT
    xPowerEnable       : BOOL; // Map to MC_Power.Enable in the axis adapter.
    xMoveVelocity      : BOOL; // Map to MC_MoveVelocity.Execute.
    xStop              : BOOL; // Map to MC_Stop.Execute.
    xReset             : BOOL; // Map to MC_Reset.Execute.
    rVelocity_mps      : REAL; // Symbolic velocity setpoint before drive scaling.
END_STRUCT
END_TYPE

TYPE ST_StationControllerConfig :
STRUCT
    rDefaultSpeed_mps       : REAL; // FDS recipe speed fallback.
    rMinimumSpeed_mps       : REAL; // Engineering lower bound.
    rMaximumSpeed_mps       : REAL; // Engineering upper bound.
    rTransitionTimeout_s    : REAL; // Generic transition watchdog for skeleton.
END_STRUCT
END_TYPE

TYPE ST_StationControllerInput :
STRUCT
    xStart             : BOOL;          // From LineSupervisor StartCell.
    xStop              : BOOL;          // From LineSupervisor StopCell.
    xReset             : BOOL;          // Reset faults/STOPPED to IDLE.
    xHold              : BOOL;          // Manual or diagnostic hold.
    xUnhold            : BOOL;          // Recover from HELD.
    xClear             : BOOL;          // Clear ABORTED to STOPPED.
    eRequestedMode     : E_PackML_Mode; // AUTO, MANUAL, MAINTENANCE.
    rTargetSpeed_mps   : REAL;          // Recipe command from supervisor.
    xSafetyLoopOK      : BOOL;          // Safety relay healthy.
    xAirPressureOK     : BOOL;          // Pneumatic pressure switch healthy.
    xVfdReady          : BOOL;          // Drive ready/no fault.
    xDiverter1Faulted  : BOOL;          // Diverter 1 diagnostic fault.
    xDiverter2Faulted  : BOOL;          // Diverter 2 diagnostic fault.
    xJamAlarm          : BOOL;          // Jam watchdog request to hold.
    xDownstreamBlocked : BOOL;          // Lane full or downstream unavailable.
    rCycleTime_s       : REAL;          // PLC task interval for unit tests.
END_STRUCT
END_TYPE

TYPE ST_StationControllerOutput :
STRUCT
    ePackMLState       : E_PackML_State;        // OPC UA ControlState.CurrentState.
    eCurrentMode       : E_PackML_Mode;         // OPC UA ControlState.CurrentMode.
    xPermissivesOK     : BOOL;                  // FDS start permissive expression.
    xRunRouting        : BOOL;                  // Enable package tracking/routing.
    xResetAlarms       : BOOL;                  // One-cycle alarm reset request.
    xConveyorRunEnable : BOOL;                  // Symbolic VFD run command.
    xConveyorQuickStop : BOOL;                  // Controlled quick stop request.
    rConveyorSpeed_mps : REAL;                  // Symbolic conveyor setpoint.
    stMotionCommand    : ST_PLCopenMotionCommand; // PLCopen command intent.
    sStatusText        : STRING(80);            // Diagnostic text.
END_STRUCT
END_TYPE

TYPE ST_StationControllerContext :
STRUCT
    eState              : E_StationControllerState;
    ePackMLState        : E_PackML_State;
    eCurrentMode        : E_PackML_Mode;
    xInitialized        : BOOL;
    xResetLast          : BOOL;
    rTransitionElapsed_s: REAL;
END_STRUCT
END_TYPE

FUNCTION F_StationController_Init : BOOL
VAR_INPUT
    stConfig : ST_StationControllerConfig;
END_VAR
VAR_IN_OUT
    stContext : ST_StationControllerContext;
    stOut     : ST_StationControllerOutput;
END_VAR

// Initialisation function. Forces the mechanical safe state.
stContext.eState := E_StationControllerState.STATION_STOPPED;
stContext.ePackMLState := E_PackML_State.STOPPED;
stContext.eCurrentMode := E_PackML_Mode.AUTO;
stContext.xInitialized := TRUE;
stContext.xResetLast := FALSE;
stContext.rTransitionElapsed_s := 0.0;

stOut.ePackMLState := E_PackML_State.STOPPED;
stOut.eCurrentMode := E_PackML_Mode.AUTO;
stOut.xPermissivesOK := FALSE;
stOut.xRunRouting := FALSE;
stOut.xResetAlarms := FALSE;
stOut.xConveyorRunEnable := FALSE;
stOut.xConveyorQuickStop := TRUE;
stOut.rConveyorSpeed_mps := 0.0;
stOut.stMotionCommand.xPowerEnable := FALSE;
stOut.stMotionCommand.xMoveVelocity := FALSE;
stOut.stMotionCommand.xStop := TRUE;
stOut.stMotionCommand.xReset := FALSE;
stOut.stMotionCommand.rVelocity_mps := 0.0;
stOut.sStatusText := 'Station controller initialised';

F_StationController_Init := TRUE;
END_FUNCTION

FUNCTION F_StationController_Cyclic : BOOL
VAR_INPUT
    stIn     : ST_StationControllerInput;
    stConfig : ST_StationControllerConfig;
END_VAR
VAR_IN_OUT
    stContext : ST_StationControllerContext;
    stOut     : ST_StationControllerOutput;
END_VAR
VAR
    xTransitionComplete : BOOL;
    rCommandSpeed_mps   : REAL;
END_VAR

// Cyclic execution function. Implements PackML sequencing with symbolic outputs.
IF stIn.rCycleTime_s > 0.0 THEN
    stContext.rTransitionElapsed_s := stContext.rTransitionElapsed_s + stIn.rCycleTime_s;
END_IF;

xTransitionComplete := stContext.rTransitionElapsed_s >= stConfig.rTransitionTimeout_s;
stOut.xResetAlarms := stIn.xReset AND NOT stContext.xResetLast;
stOut.xPermissivesOK := stIn.xSafetyLoopOK
                        AND stIn.xAirPressureOK
                        AND stIn.xVfdReady
                        AND NOT stIn.xDiverter1Faulted
                        AND NOT stIn.xDiverter2Faulted;

rCommandSpeed_mps := stIn.rTargetSpeed_mps;
IF rCommandSpeed_mps < stConfig.rMinimumSpeed_mps THEN
    rCommandSpeed_mps := stConfig.rDefaultSpeed_mps;
END_IF;
IF rCommandSpeed_mps > stConfig.rMaximumSpeed_mps THEN
    rCommandSpeed_mps := stConfig.rMaximumSpeed_mps;
END_IF;

IF NOT stContext.xInitialized THEN
    stContext.eState := E_StationControllerState.STATION_UNINITIALISED;
    stContext.ePackMLState := E_PackML_State.STOPPED;
ELSIF NOT stIn.xSafetyLoopOK THEN
    stContext.eState := E_StationControllerState.STATION_ABORTED;
    stContext.ePackMLState := E_PackML_State.ABORTED;
    stContext.rTransitionElapsed_s := 0.0;
ELSE
    CASE stContext.ePackMLState OF
        E_PackML_State.STOPPED:
            stContext.eState := E_StationControllerState.STATION_STOPPED;
            IF stIn.xReset THEN
                stContext.ePackMLState := E_PackML_State.RESETTING;
                stContext.rTransitionElapsed_s := 0.0;
            END_IF;

        E_PackML_State.RESETTING:
            stContext.eState := E_StationControllerState.STATION_RESETTING;
            IF xTransitionComplete THEN
                stContext.ePackMLState := E_PackML_State.IDLE;
                stContext.rTransitionElapsed_s := 0.0;
            END_IF;

        E_PackML_State.IDLE:
            stContext.eState := E_StationControllerState.STATION_IDLE;
            IF stIn.xStop THEN
                stContext.ePackMLState := E_PackML_State.STOPPING;
                stContext.rTransitionElapsed_s := 0.0;
            ELSIF stIn.xStart AND stOut.xPermissivesOK THEN
                stContext.ePackMLState := E_PackML_State.STARTING;
                stContext.rTransitionElapsed_s := 0.0;
            END_IF;

        E_PackML_State.STARTING:
            stContext.eState := E_StationControllerState.STATION_STARTING;
            IF stIn.xStop THEN
                stContext.ePackMLState := E_PackML_State.STOPPING;
                stContext.rTransitionElapsed_s := 0.0;
            ELSIF xTransitionComplete AND stOut.xPermissivesOK THEN
                stContext.ePackMLState := E_PackML_State.EXECUTE;
                stContext.rTransitionElapsed_s := 0.0;
            END_IF;

        E_PackML_State.EXECUTE:
            stContext.eState := E_StationControllerState.STATION_EXECUTE;
            IF stIn.xStop THEN
                stContext.ePackMLState := E_PackML_State.STOPPING;
                stContext.rTransitionElapsed_s := 0.0;
            ELSIF stIn.xJamAlarm OR stIn.xHold OR NOT stOut.xPermissivesOK THEN
                stContext.ePackMLState := E_PackML_State.HOLDING;
                stContext.rTransitionElapsed_s := 0.0;
            ELSIF stIn.xDownstreamBlocked THEN
                stContext.ePackMLState := E_PackML_State.SUSPENDED;
                stContext.rTransitionElapsed_s := 0.0;
            END_IF;

        E_PackML_State.SUSPENDED:
            stContext.eState := E_StationControllerState.STATION_SUSPENDED;
            IF stIn.xStop THEN
                stContext.ePackMLState := E_PackML_State.STOPPING;
                stContext.rTransitionElapsed_s := 0.0;
            ELSIF NOT stIn.xDownstreamBlocked THEN
                stContext.ePackMLState := E_PackML_State.EXECUTE;
                stContext.rTransitionElapsed_s := 0.0;
            END_IF;

        E_PackML_State.HOLDING:
            stContext.eState := E_StationControllerState.STATION_HOLDING;
            IF xTransitionComplete THEN
                stContext.ePackMLState := E_PackML_State.HELD;
                stContext.rTransitionElapsed_s := 0.0;
            END_IF;

        E_PackML_State.HELD:
            stContext.eState := E_StationControllerState.STATION_HELD;
            IF stIn.xStop THEN
                stContext.ePackMLState := E_PackML_State.STOPPING;
                stContext.rTransitionElapsed_s := 0.0;
            ELSIF stIn.xUnhold AND stOut.xPermissivesOK AND NOT stIn.xJamAlarm THEN
                stContext.ePackMLState := E_PackML_State.UNHOLDING;
                stContext.rTransitionElapsed_s := 0.0;
            END_IF;

        E_PackML_State.UNHOLDING:
            stContext.eState := E_StationControllerState.STATION_UNHOLDING;
            IF stIn.xStop THEN
                stContext.ePackMLState := E_PackML_State.STOPPING;
                stContext.rTransitionElapsed_s := 0.0;
            ELSIF xTransitionComplete THEN
                stContext.ePackMLState := E_PackML_State.EXECUTE;
                stContext.rTransitionElapsed_s := 0.0;
            END_IF;

        E_PackML_State.STOPPING:
            stContext.eState := E_StationControllerState.STATION_STOPPING;
            IF xTransitionComplete THEN
                stContext.ePackMLState := E_PackML_State.STOPPED;
                stContext.rTransitionElapsed_s := 0.0;
            END_IF;

        E_PackML_State.ABORTED:
            stContext.eState := E_StationControllerState.STATION_ABORTED;
            IF stIn.xClear THEN
                stContext.ePackMLState := E_PackML_State.STOPPED;
                stContext.rTransitionElapsed_s := 0.0;
            END_IF;
    END_CASE;
END_IF;

IF (stContext.ePackMLState = E_PackML_State.STOPPED)
   OR (stContext.ePackMLState = E_PackML_State.IDLE)
   OR (stContext.ePackMLState = E_PackML_State.ABORTED) THEN
    stContext.eCurrentMode := stIn.eRequestedMode;
END_IF;

stOut.ePackMLState := stContext.ePackMLState;
stOut.eCurrentMode := stContext.eCurrentMode;
stOut.xRunRouting := stContext.ePackMLState = E_PackML_State.EXECUTE;
stOut.xConveyorRunEnable := (stContext.ePackMLState = E_PackML_State.STARTING)
                            OR (stContext.ePackMLState = E_PackML_State.EXECUTE)
                            OR (stContext.ePackMLState = E_PackML_State.UNHOLDING);
stOut.xConveyorQuickStop := (stContext.ePackMLState = E_PackML_State.HOLDING)
                            OR (stContext.ePackMLState = E_PackML_State.HELD)
                            OR (stContext.ePackMLState = E_PackML_State.ABORTED)
                            OR (stContext.ePackMLState = E_PackML_State.STOPPING);

IF stOut.xConveyorRunEnable THEN
    stOut.rConveyorSpeed_mps := rCommandSpeed_mps;
ELSE
    stOut.rConveyorSpeed_mps := 0.0;
END_IF;

// PLCopen motion sequence intent; a target-specific adapter binds these to MC_* FBs.
stOut.stMotionCommand.xPowerEnable := stOut.xPermissivesOK AND (stContext.ePackMLState <> E_PackML_State.ABORTED);
stOut.stMotionCommand.xMoveVelocity := stOut.xConveyorRunEnable;
stOut.stMotionCommand.xStop := stOut.xConveyorQuickStop;
stOut.stMotionCommand.xReset := stOut.xResetAlarms;
stOut.stMotionCommand.rVelocity_mps := stOut.rConveyorSpeed_mps;
stOut.sStatusText := 'Station PackML sequence evaluated';

stContext.xResetLast := stIn.xReset;
F_StationController_Cyclic := stContext.xInitialized;
END_FUNCTION

FUNCTION_BLOCK FB_StationController
VAR_INPUT
    stIn     : ST_StationControllerInput;  // Typed symbolic inputs.
    stConfig : ST_StationControllerConfig; // Testable configuration.
    xInit    : BOOL;                       // Pulse to re-run initialisation.
END_VAR
VAR_OUTPUT
    stOut        : ST_StationControllerOutput; // Typed symbolic outputs.
    eState       : E_StationControllerState;   // Exposed module state.
    xInitialized : BOOL;                       // Module initialisation complete.
END_VAR
VAR
    stContext : ST_StationControllerContext;
    xInitLast : BOOL;
END_VAR

IF (NOT stContext.xInitialized) OR (xInit AND NOT xInitLast) THEN
    F_StationController_Init(stConfig := stConfig, stContext := stContext, stOut := stOut);
END_IF;

F_StationController_Cyclic(stIn := stIn, stConfig := stConfig, stContext := stContext, stOut := stOut);

eState := stContext.eState;
xInitialized := stContext.xInitialized;
xInitLast := xInit;
END_FUNCTION_BLOCK
